# EPICS substitutions: db/ecat2el4104.substitutions
file ecat2el41xx.template
{
	pattern {CH_ID, PDO_IDX, EOFF, ESLO}
		{$(MOD_ID)-AO1, 0, 0, 0.0003051850947599719}
		{$(MOD_ID)-AO2, 1, 0, 0.0003051850947599719}
		{$(MOD_ID)-AO3, 2, 0, 0.0003051850947599719}
		{$(MOD_ID)-AO4, 3, 0, 0.0003051850947599719}
}

file ecat2slave.template
{
	pattern {DTYP}
		{EL4104}
}
